INTERFACE I_Base

END_INTERFACE

(* stored: Version 1.1.0.1
   Itf I_Base: Id {77777777-7777-7777-7777-777777777702} *)
